{attribute 'qualified_only'}
{attribute 'strict'}
{attribute 'to_string'}
TYPE E_DS402MotionMode :
(
    DISCRETE := 0,
    CONTINUOUS := 1,
    SYNCHRONOUS := 2
) UINT;
END_TYPE

(* stored: Version 1.1.0.1
   DUT E_DS402MotionMode: Id {38aa60c9-8af6-4ab2-8e1c-de410c7e8e23} *)
